TYPE (* IEC61131-3, Table 14#5 *)
  (* Standard: 1131-3 *)
  (* Version 0.0, 1/8/2024, Cheyan, Schneider Electric, Template *)
  PACKAGE Main;
  {SET_ATTRIBUTE(nxtDataType, CJbEgK4hJZ+OVMCPag09+k0G/MZnYfwme0Gl/B4lr0bVvPw4cKa3j72fUQKXk2XAxPBvjuSeEkHtp3D/XZYMaqoqrnj7hb1AjWzfbIHWL6wNRN+ztk1GPMuoHUnUV0PyIQMdJ6w2weBBNy6h+x+ZMPlXDJNYnrXfh8riE9KyGcNkJQYcKScB5z5Z2slviNsjRvjdhv8ErLQ=)}
  CtlModels : (
    item1,
    item2,
    item3
  );
END_TYPE
